# EPICS autosave request: iocBoot/gmca_23b_ioc2/dbSave/auto_positions.req
#
 23b:2:scan1.VAL

file bluice.req P=23b:
